FUNCTION TryConvert_UDINT_TO_INT : BOOL
VAR_INPUT
	in : UDINT;
	out : REFERENCE TO INT;
END_VAR

IF in > DatatypeLimits.MAX_VALUE_OF_UDINT_WHICH_CAN_BE_HELD_IN_A_INT THEN
	RETURN;
END_IF

out := UDINT_TO_INT(in);
TryConvert_UDINT_TO_INT := TRUE;

END_FUNCTION

(* stored: Version 1.1.0.1, ProductVersion 3.1.4024.12
   POU TryConvert_UDINT_TO_INT: Id {3fb4860d-2aae-4b48-b9f5-42249b9bc5cd}, SpecialFunc None *)
